// TwinCAT 3 PLC project XY_Motion_Control
// ProgramVersion: 3.1.4024.0
// libraries:
//   Tc2_Math, * (Beckhoff Automation GmbH)
//   Tc2_MC2, * (Beckhoff Automation GmbH)
//   Tc2_Standard, * (Beckhoff Automation GmbH)
//   Tc2_System, * (Beckhoff Automation GmbH)
//   Tc3_Module, * (Beckhoff Automation GmbH)
// project tree:
//   DUTs/ E_AutoSeqState.TcDUT, ST_MotionStep.TcDUT
//   / GlobalTextList.TcGTLO, PlcTask.TcTTO, Visualization Manager.TcVMO (not stored)
//   GVLs/ GVL_Motion.TcGVL
//   POUs/ AutoSequence.TcPOU, FB_XYZ_Movement.TcPOU, MAIN.TcPOU
//   VISUs/ Visualization.TcVIS
// real-time tasks:
//   TASK PlcTask: cycle T#10ms, priority 20, ADS port 350
// motion (NC):
//   TASK NC-Task 1 SAF: cycle T#2ms, priority 4, ADS port 501
//   TASK NC-Task 1 SVB: cycle T#10ms, priority 8, ADS port 511
//   AXIS Axis 1 (X) (id 1) // This is the X axis
//     Velo: RefSearch=3, SlowManual=5, FastManual=50
//     OtherSettings: AllowMotionCmdToSlave=true
//     encoder EncType=19
//       EncPara: ScaleFactorNumerator=3.8147e-05, MaxCount=#xffffffff
//         SoftEndMinControl: Enable=true, Range=-0.1
//         SoftEndMaxControl: Enable=true, Range=9.9
//         Inc: RefSoftSyncMask=#xffffffff
//     drive DrvType=16
//       DrvPara: MaxCount=#xffffffff, DriveControlDWord=#x00020100
//         Analog: TorqueSetpointScale=10, ScaleFactorActTorque=0.1
//         TimeComp: TaskDelayCycles=1
//     controller CtrType=1
//       CtrPara: PriorControlFactor=1
//         Observer: BandWidth=20
//   AXIS Axis 2 (Y) (id 2) // This is the Y axis
//     Velo: RefSearch=3, SlowManual=10, FastManual=50
//     OtherSettings: AllowMotionCmdToSlave=true
//     encoder EncType=19
//       EncPara: MaxCount=#xffffffff
//         SoftEndMinControl: Enable=true, Range=-34
//         SoftEndMaxControl: Enable=true
//         Inc: RefSoftSyncMask=#xffffffff
//     drive DrvType=16
//       DrvPara: MaxCount=#xffffffff, DriveControlDWord=#x00020100
//         Analog: TorqueSetpointScale=10, ScaleFactorActTorque=0.1
//         TimeComp: TaskDelayCycles=1
//     controller CtrType=1
//       CtrPara: PriorControlFactor=1
//         Observer: BandWidth=20
// I/O:
//   DEVICE Device 1 (Profinet Device CCAT (RT)) (disabled), AmsNetId 5.55.247.106.2.1
//   DEVICE Device 2 (EtherCAT), AmsNetId 5.55.247.106.3.1
//     Term 1 (EK1200) [EK1200-5000 EtherCAT Power supply (2A E-Bus)]
//       Term 2 (EL1008) [EL1008 8Ch. Dig. Input 24V, 3ms]
//       Term 3 (EL2008) [EL2008 8Ch. Dig. Output 24V, 0.5A]
//       Term 4 (EL9011) [EL9011 End Terminal]
//   DEVICE Device 5 (EtherCAT), AmsNetId 5.55.247.106.6.1
//     Drive 5 (R88D-KN01H-ECT) [R88D-KN01H-ECT G5 Series ServoDrive/Motor]
//     Drive 6 (R88D-KN01H-ECT) [R88D-KN01H-ECT G5 Series ServoDrive/Motor]
//   DEVICE Device 3 (NOV-DP-RAM)
// variable links:
//   NC-Task 1 SAF/Axes/Axis 1 (X) <-> Device 5 (EtherCAT)/Drive 5 (R88D-KN01H-ECT)
//     Drive/Inputs/In/nDataIn1 <-> 258th transmit PDO Mapping/Following error actual value
//     Drive/Inputs/In/nDataIn3[0] <-> 258th transmit PDO Mapping/Torque actual value
//     Drive/Inputs/In/nDcOutputTime <-> InfoData/DcOutputShift
//     Drive/Inputs/In/nState1 <-> 258th transmit PDO Mapping/Statusword
//     Drive/Inputs/In/nState2 <-> 258th transmit PDO Mapping/Statusword @bit 8
//     Drive/Inputs/In/nState4 @bit 1 <-> WcState/InputToggle
//     Drive/Inputs/In/nState4 <-> WcState/WcState
//     Drive/Outputs/Out/nCtrl1 <-> 258th receive PDO Mapping/Controlword
//     Drive/Outputs/Out/nCtrl2 <-> 258th receive PDO Mapping/Controlword @bit 8
//     Drive/Outputs/Out/nDataOut1 <-> 258th receive PDO Mapping/Target position
//     Enc/Inputs/In/nDataIn1 <-> 258th transmit PDO Mapping/Position actual value
//     Enc/Inputs/In/nDataIn3 <-> 258th transmit PDO Mapping/Touch probe pos1 pos value
//     Enc/Inputs/In/nDataIn5 <-> 258th transmit PDO Mapping/Touch probe pos2 pos value
//     Enc/Inputs/In/nDcInputTime <-> InfoData/DcInputShift
//     Enc/Inputs/In/nState4 @bit 1 <-> WcState/InputToggle
//     Enc/Inputs/In/nState4 <-> WcState/WcState
//     Enc/Inputs/In/nState5 <-> 258th transmit PDO Mapping/Touch probe status
//     Enc/Inputs/In/nState6 <-> 258th transmit PDO Mapping/Touch probe status @bit 8
//     Enc/Outputs/Out/nCtrl5 <-> 258th receive PDO Mapping/Touch probe function
//     Enc/Outputs/Out/nCtrl6 <-> 258th receive PDO Mapping/Touch probe function @bit 8
//   NC-Task 1 SAF/Axes/Axis 2 (Y) <-> Device 5 (EtherCAT)/Drive 6 (R88D-KN01H-ECT)
//     Drive/Inputs/In/nDataIn1 <-> 258th transmit PDO Mapping/Following error actual value
//     Drive/Inputs/In/nDataIn3[0] <-> 258th transmit PDO Mapping/Torque actual value
//     Drive/Inputs/In/nDcOutputTime <-> InfoData/DcOutputShift
//     Drive/Inputs/In/nState1 <-> 258th transmit PDO Mapping/Statusword
//     Drive/Inputs/In/nState2 <-> 258th transmit PDO Mapping/Statusword @bit 8
//     Drive/Inputs/In/nState4 @bit 1 <-> WcState/InputToggle
//     Drive/Inputs/In/nState4 <-> WcState/WcState
//     Drive/Outputs/Out/nCtrl1 <-> 258th receive PDO Mapping/Controlword
//     Drive/Outputs/Out/nCtrl2 <-> 258th receive PDO Mapping/Controlword @bit 8
//     Drive/Outputs/Out/nDataOut1 <-> 258th receive PDO Mapping/Target position
//     Enc/Inputs/In/nDataIn1 <-> 258th transmit PDO Mapping/Position actual value
//     Enc/Inputs/In/nDataIn3 <-> 258th transmit PDO Mapping/Touch probe pos1 pos value
//     Enc/Inputs/In/nDataIn5 <-> 258th transmit PDO Mapping/Touch probe pos2 pos value
//     Enc/Inputs/In/nDcInputTime <-> InfoData/DcInputShift
//     Enc/Inputs/In/nState4 @bit 1 <-> WcState/InputToggle
//     Enc/Inputs/In/nState4 <-> WcState/WcState
//     Enc/Inputs/In/nState5 <-> 258th transmit PDO Mapping/Touch probe status
//     Enc/Inputs/In/nState6 <-> 258th transmit PDO Mapping/Touch probe status @bit 8
//     Enc/Outputs/Out/nCtrl5 <-> 258th receive PDO Mapping/Touch probe function
//     Enc/Outputs/Out/nCtrl6 <-> 258th receive PDO Mapping/Touch probe function @bit 8
//   XY_Motion_Control/Motion_Control <-> Device 2 (EtherCAT)/Term 1 (EK1200)/Term 2 (EL1008)
//     PlcTask Inputs/GVL_Motion.bSensor_X <-> Channel 1/Input
//     PlcTask Inputs/GVL_Motion.bSensor_Y <-> Channel 3/Input
//   XY_Motion_Control/Motion_Control <-> Device 2 (EtherCAT)/Term 1 (EK1200)/Term 3 (EL2008)
//     PlcTask Outputs/GVL_Motion.bZlifter <-> Channel 2/Output
//   XY_Motion_Control/Motion_Control <-> NC-Task 1 SAF/Axes/Axis 1 (X)
//     PlcTask Inputs/GVL_Motion.Axis1.NcToPlc <-> Outputs/ToPlc
//     PlcTask Outputs/GVL_Motion.Axis1.PlcToNc <-> Inputs/FromPlc
//   XY_Motion_Control/Motion_Control <-> NC-Task 1 SAF/Axes/Axis 2 (Y)
//     PlcTask Inputs/GVL_Motion.Axis2.NcToPlc <-> Outputs/ToPlc
//     PlcTask Outputs/GVL_Motion.Axis2.PlcToNc <-> Inputs/FromPlc

CONFIGURATION XY_Motion_Control
    RESOURCE PLC ON TwinCAT3
        TASK PlcTask(INTERVAL := T#10ms, PRIORITY := 20);
        PROGRAM MAIN WITH PlcTask : MAIN;
    END_RESOURCE
END_CONFIGURATION

// ---- DUTs/E_AutoSeqState.TcDUT
{attribute 'qualified_only'}
{attribute 'strict'}
// Moves for the auto sequence
// Auto sekvenssin liikkeet
TYPE E_AutoSeqState :
(
	INIT,
    MOVE_X_SAFE_HOME,
	WAIT_X_SAFE_HOME,

    SET_Z_POSITION,
    WAIT_Z_DELAY,

    DECIDE_MOVE_ORDER,
	MOVE_Y,
    WAIT_Y,

    MOVE_X,
    WAIT_X,

    NEXT_STEP,

    PREPARE_RETURN_HOME,
    RETURN_HOME

);
END_TYPE

// ---- DUTs/ST_MotionStep.TcDUT
TYPE ST_MotionStep :
STRUCT
	fTargetX		: LREAL; // Target position of X axis - AXIS1, X axis kohde asento
	fTargetY		: LREAL; // Target position of Y axis - AXIS2, Y axis kohde asento
	nZaction		: INT; 	 // 1 = Lift, 2 = Lower, 0 = Do nothing, nostimen asennot
END_STRUCT
END_TYPE

// ---- GVLs/GVL_Motion.TcGVL
{attribute 'qualified_only'}
{attribute 'qualified_only'}
VAR_GLOBAL
	// Author RL
	// Hardware axis references
	// Axis viittaukset
	Axis1               : AXIS_REF;	// X
	Axis2               : AXIS_REF;	// Y
	
	// Core system control
	bEnableAll          : BOOL := TRUE;		// Enables the servo drives, aktivoi servot
	bResetAll           : BOOL := FALSE;	// Resets possible servo errors, resetoi servo viat
	bManualModeActive   : BOOL := FALSE; 	// Enables manual driving, aktivoi manualiajon
	
	// Homing inputs and status check after homing
	// Kotiutus inputit ja tarkistus kotiutuksen jälkeen
	bSensor_X           AT %I* : BOOL; 
	bSensor_Y           AT %I* : BOOL;
	bStartHoming        : BOOL := FALSE; 
	bXHomed             : BOOL := FALSE; 
	bYHomed             : BOOL := FALSE; 

	// Live axis position
	// Live axis asennot
	fCurrentX           : LREAL := 0.0;
	fCurrentY           : LREAL := 0.0;

	// "Z Axis" not really but kinda acts as a Z axis, this is a pneumatic lifter that is sitting on the Y axis
	// "Z Axis" Paineilma nostin Y akselin päällä
	bZlifter            AT %Q* : BOOL;      // FALSE = Raised, TRUE = Lowered)
	bZlifterManual		: BOOL;
	
	// Controls for manual driving, "Jogging"
	// Manuaaliajon kontrollit
	bJogForwardX        : BOOL := FALSE;    
	bJogForwardY        : BOOL := FALSE;    
	bJogBackwardsX      : BOOL := FALSE;    
	bJogBackwardsY      : BOOL := FALSE;
	fVelocityX          : LREAL := 5.0;
	fVelocityY          : LREAL := 10.0;
	
	// These calculate if moving is allowed, based on current position
	// Liikkumisen luvat, nykyisen sijainnin mukaan
	bX_Allow_Positive   : BOOL := FALSE;
	bX_Allow_Negative   : BOOL := FALSE;
	bY_Allow_Positive   : BOOL := FALSE;
	bY_Allow_Negative   : BOOL := FALSE;
	
	// States
	// Z nostimen tilat
	Z_IDLE          : INT := 0;
	Z_UP            : INT := 1;
	Z_DOWN          : INT := 2;
	
	iAutoState          : INT := 0; 
	bStartAutoseq     	: BOOL := FALSE;
	bAutoseqDone     	: BOOL := FALSE;
	bSequenceRunning	: BOOL;
	bRetrievalMode    	: BOOL := FALSE;  // FALSE = Put away pallets, TRUE = Take away pallets / Autosekvenssin Z lifter käänteiset tilat
	
	bExecuteMoveX    : BOOL;
    bExecuteMoveY    : BOOL;
    fTargetX         : LREAL;
    fTargetY         : LREAL;

	
	iStepPointer        : INT := 1;
	eSubPhase           : E_AutoSeqState := E_AutoSeqState.INIT;
	iTotalSteps         : INT := 9;
	
	// Go to config if u change these settings
	// This array system holds inside coordinates for the automatic sequence driving
	// Actions of the pneumatic lift are reversed when bRetrievalMode = TRUE
	// Automaattisen sekvenssin koordinaatit
	// Lifterin aktionit päinvaistaiset kun bRetrievalMode = TRUE
	astPath : ARRAY[1..9] OF ST_MotionStep := [
		// "Shelf 1" cycle
		
		(fTargetX := 2.8000, fTargetY := -0.6247,  nZAction := 1), // 2. Moce Y to shelf 1 height
		(fTargetX := 9.3720, fTargetY := -0.6247,  nZAction := 2), // 3. Drive in and lower forks
		(fTargetX := 2.8000, fTargetY := -0.6247,  nZAction := 1), // 4. Retreat to safe line and raise forks
		
		// "Shelf 2" cycle
		(fTargetX := 2.8000, fTargetY := -9.5381,	nZAction := 0), // 5. Drop Y to shelf 2 height
		(fTargetX := 9.3720, fTargetY := -9.5381,	nZAction := 2), // 6. Drive in and lower forks
		(fTargetX := 2.8000, fTargetY := -9.5381,	nZAction := 1), // 7. Retreat to safe line and raise forks
		
		// "Shelf 3" cycle
		(fTargetX := 2.8000, fTargetY := -18.7514,	nZAction := 0), // 8. Drop Y to shelf 3 height
		(fTargetX := 9.3720, fTargetY := -18.7514,	nZAction := 2), // 9. Drive in and lower forks
		(fTargetX := 0.0,	 fTargetY := -18.7514,	nZAction := 1)	// 10. Drive X out to 0 keep Y still
		
		
		// The auto sequence automatically handles moving X and Y back to 0.0 after this step	
	];
	
END_VAR

// ---- POUs/MAIN.TcPOU
// Author RL
PROGRAM MAIN
VAR
	XYZ	: FB_XYZ_Movement;
END_VAR

// Execute the entire system
AutoSequence();

XYZ(Axis1 := GVL_Motion.Axis1, Axis2 := GVL_Motion.Axis2);

END_PROGRAM

// ---- POUs/FB_XYZ_Movement.TcPOU
FUNCTION_BLOCK FB_XYZ_Movement
VAR_IN_OUT
    // Axis references
    Axis1                : AXIS_REF; // X
    Axis2                : AXIS_REF; // Y
END_VAR
VAR
    // Hardware Power and Reset Blocks
    fbPower1             : MC_Power;
    fbPower2             : MC_Power;
	
    fbReset1             : MC_Reset;
    fbReset2             : MC_Reset;
    
    // Core Motion Instances
    fbAutoMoveX          : MC_MoveAbsolute;
    fbAutoMoveY          : MC_MoveAbsolute;
	
    fbDriveToSensorX     : MC_MoveVelocity;
    fbDriveToSensorY     : MC_MoveVelocity;
	
    fbStopX              : MC_Stop;
    fbStopY              : MC_Stop;
	
    fbLockZeroX          : MC_SetPosition;
    fbLockZeroY          : MC_SetPosition;
	
    fbJogX               : MC_Jog;
    fbJogY               : MC_Jog;
	
	//Safety position reference
	fActPosX				 : LREAL;
	fActPosY				 : LREAL;
END_VAR

// Safety first, position reference form axis
// Paikan haku
fActPosX	:= Axis1.NcToPlc.ActPos;
fActPosY	:= Axis2.NcToPlc.ActPos;
THIS^.M_UpdateSafety();

// Axis Power, directional enables based on position
// Axis teho, luvat liike suunnille sijainnin perusteella
// X Axis 1
fbPower1(
    Axis            := Axis1, 
    Enable          := GVL_Motion.bEnableAll, 
    Enable_Positive := GVL_Motion.bEnableAll AND GVL_Motion.bX_Allow_Positive, 
    Enable_Negative := GVL_Motion.bEnableAll AND GVL_Motion.bX_Allow_Negative
);
// Y Axis 2
fbPower2(
    Axis            := Axis2, 
    Enable          := GVL_Motion.bEnableAll, 
    Enable_Positive := GVL_Motion.bEnableAll AND GVL_Motion.bY_Allow_Positive, 
    Enable_Negative := GVL_Motion.bEnableAll AND GVL_Motion.bY_Allow_Negative
);

// NC Kernel Error Resets
// Axis error resetit
fbReset1(
	Axis := Axis1,
	Execute := GVL_Motion.bResetAll);
	
fbReset2(
	Axis := Axis2,
	Execute := GVL_Motion.bResetAll);

IF GVL_Motion.bResetAll THEN
    GVL_Motion.bResetAll := FALSE;
END_IF

// Automated sequence, axis ref and enables, edit velocity if needed
// Automaattisen sekvenssin, axis viittaus ja luvat, tästä voi muutta automaattisen sekvenssin nopeutta halutessa
// Jos nopeutta on liikaa servo menee error tilaan (Set point karkaa liian kauas)
fbAutoMoveX(
    Axis     := Axis1, 
    Execute  := GVL_Motion.bExecuteMoveX AND NOT GVL_Motion.bManualModeActive, 
    Position := GVL_Motion.fTargetX, 
    Velocity := 10.0
);

fbAutoMoveY(
    Axis     := Axis2, 
    Execute  := GVL_Motion.bExecuteMoveY AND NOT GVL_Motion.bManualModeActive, 
    Position := GVL_Motion.fTargetY, 
    Velocity := 20.0
);


// Manual control, axis ref and enables
// Manuaali ajon axis viittaus, luvat
fbJogX(
    Axis         := Axis1,
    JogForward   := GVL_Motion.bJogForwardX AND GVL_Motion.bX_Allow_Positive AND GVL_Motion.bManualModeActive AND NOT GVL_Motion.bStartAutoseq,
    JogBackwards := GVL_Motion.bJogBackwardsX AND GVL_Motion.bX_Allow_Negative AND GVL_Motion.bManualModeActive AND NOT GVL_Motion.bStartAutoseq,
    Mode         := MC_JOGMODE_CONTINOUS,
    Velocity     := GVL_Motion.fVelocityX
);

fbJogY(
    Axis         := Axis2,
    JogForward   := GVL_Motion.bJogForwardY AND GVL_Motion.bY_Allow_Positive AND GVL_Motion.bManualModeActive AND NOT GVL_Motion.bStartAutoseq,
    JogBackwards := GVL_Motion.bJogBackwardsY AND GVL_Motion.bY_Allow_Negative AND GVL_Motion.bManualModeActive AND NOT GVL_Motion.bStartAutoseq,
    Mode         := MC_JOGMODE_CONTINOUS,
    Velocity     := GVL_Motion.fVelocityY
);

// Safety reset to turn off manual jogging if switched away from manual mode
// Manualiset liike komennot lakkaa, jos vaihdetaan kesken kaiken pois manuaali tilasta
IF NOT GVL_Motion.bManualModeActive THEN
    fbJogX(
		Axis := Axis1,
		JogForward := FALSE,
		JogBackwards := FALSE);
		
    fbJogY(
		Axis := Axis2,
		JogForward := FALSE,
		JogBackwards := FALSE);
END_IF

// Homing
// Kotiutus
fbDriveToSensorX(
	Axis := Axis1,
	Execute := GVL_Motion.bStartHoming,
	Velocity := 5.0,
	Direction := MC_Negative_Direction);
	
fbStopX(
	Axis := Axis1,
	Execute := GVL_Motion.bStartHoming AND GVL_Motion.bSensor_X);
	
fbLockZeroX(
	Axis := Axis1,
	Execute := GVL_Motion.bStartHoming AND fbStopX.Done,
	Position := 0.0);

fbDriveToSensorY(
	Axis := Axis2,
	Execute := GVL_Motion.bStartHoming,
	Velocity := 17.0,
	Direction := MC_Positive_Direction);
	
fbStopY(
	Axis := Axis2,
	Execute := GVL_Motion.bStartHoming AND GVL_Motion.bSensor_Y);
	
fbLockZeroY(
	Axis := Axis2,
	Execute := GVL_Motion.bStartHoming AND fbStopY.Done,
	Position := 0.0);

// Homing indication
// Kotiutuksen indikointi
IF fbLockZeroX.Done THEN 
    GVL_Motion.bXHomed := TRUE;
END_IF

IF fbLockZeroY.Done THEN
    GVL_Motion.bYHomed := TRUE;
END_IF

// Reset Homing when done
// Resetoidaan kotiutus kun se on valmis
IF GVL_Motion.bXHomed AND GVL_Motion.bYHomed THEN
    GVL_Motion.bStartHoming := FALSE;
END_IF

// Reset homing executions, so that homing can be done again if needed
// Resetoidaan kotiutus, jos tarvitaan uudestaan kotiuttaa
IF NOT GVL_Motion.bStartHoming THEN
    fbDriveToSensorX(
		Axis := Axis1,
		Execute := FALSE);
		
    fbStopX(
		Axis := Axis1,
		Execute := FALSE);
		
    fbLockZeroX(
		Axis := Axis1,
		Execute := FALSE);
    
    fbDriveToSensorY(
		Axis := Axis2,
		Execute := FALSE);
    
	fbStopY(
		Axis := Axis2, 
		Execute := FALSE);
    
	fbLockZeroY(
		Axis := Axis2,
		Execute := FALSE);
END_IF

// Author RL
METHOD PRIVATE M_UpdateSafety
VAR_INPUT
END_VAR
//Author RL
// System position
// Systeemin sijainti
GVL_Motion.fCurrentX := fActPosX;
GVL_Motion.fCurrentY := fActPosY;

IF GVL_Motion.bSequenceRunning THEN
    GVL_Motion.bManualModeActive := FALSE;
END_IF

IF GVL_Motion.bStartHoming THEN
    // During homing all movement is allowed
	// Kotiutuksen aikana kaikki liikesuunnan sallittu
    GVL_Motion.bX_Allow_Negative := TRUE; 
    GVL_Motion.bX_Allow_Positive := TRUE;
    GVL_Motion.bY_Allow_Negative := TRUE; 
    GVL_Motion.bY_Allow_Positive := TRUE;
END_IF
	
IF GVL_Motion.bManualModeActive THEN
	// Different safety limits for manual driving, this is to prevent hitting the shelves with forks in manual mode.
	// These are editable from here, but not recommended to ensure safe operation
	// Manuaaliajolla eri turvarajat, voi muutta, mutta ei suositeltu
	GVL_Motion.bX_Allow_Negative := (GVL_Motion.fCurrentX > -0.1);
    GVL_Motion.bX_Allow_Positive := (GVL_Motion.fCurrentX < 5.820);	// Note X is allowed to travell less in manual to protect possible forks/ Z lifter
                                       
    GVL_Motion.bY_Allow_Negative := (GVL_Motion.fCurrentY > -34.0);
   	GVL_Motion.bY_Allow_Positive := (GVL_Motion.fCurrentY < 0.0);
	
	GVL_Motion.bZlifter := GVL_Motion.bZlifterManual;	// Manual control for Z lifter, manuaaliset kontrollit Z lifterille
END_IF

IF GVL_Motion.bSequenceRunning THEN
	// Safety limits for automatic sequence
	// These same values are also in the AXIS settings under parameter - limit switches
	// These values are safe operation boundaries so that we dont crash the lifter/forks in to the shelves
	// If you wish to edit these, go under Axis -> Parameters -> Limit switches
	// Auto sekvenssin turvarajat, nämä on myös asetettu suoraan molempiin Axiksiin niiden asetuksista
    GVL_Motion.bX_Allow_Negative := (GVL_Motion.fCurrentX > -0.1);
    GVL_Motion.bX_Allow_Positive := (GVL_Motion.fCurrentX < 9.9);
                                        
    GVL_Motion.bY_Allow_Negative := (GVL_Motion.fCurrentY > -34.0);
    GVL_Motion.bY_Allow_Positive := (GVL_Motion.fCurrentY < 0.0);
END_IF
END_METHOD

END_FUNCTION_BLOCK

// ---- POUs/AutoSequence.TcPOU
// Author RL
PROGRAM AutoSequence
VAR
    bSequenceResetPulse : BOOL;
    tPneumaticDelay     : TON;
    bOldZlifter         : BOOL;
	bSequenceRunning	: BOOL;
END_VAR

// Author RL
IF GVL_Motion.bStartAutoseq AND GVL_Motion.bXHomed AND GVL_Motion.bYHomed AND NOT GVL_Motion.bSequenceRunning THEN
    GVL_Motion.bStartAutoseq    := FALSE; // Switches HMI button to FALSE, Laittaa HMI nappulan FALSE
    GVL_Motion.bSequenceRunning := TRUE;  // True while sequence running, TRUE kun sekvenssi käynnissä
    GVL_Motion.bAutoseqDone     := FALSE; // FALSE while sequence active, FALSE kun sekvenssi käynnissä
	
	GVL_Motion.iStepPointer     := 1;     
    GVL_Motion.bExecuteMoveX    := FALSE; // Wipes old move triggers, pyyhkii vanhat executet
    GVL_Motion.bExecuteMoveY    := FALSE; // Wipes old move triggers, pyyhkii vanhat executet
	
    GVL_Motion.eSubPhase		:= E_AutoSeqState.INIT;
	
END_IF

// Auto Sequence / Automaattinen sekvenssi
IF GVL_Motion.bSequenceRunning THEN
    bSequenceResetPulse := FALSE;

    // Check if there are still valid steps left to run in path array
    // Tarkastetaan onko vielä askelia jäljellä
    IF GVL_Motion.iStepPointer <= GVL_Motion.iTotalSteps THEN
    
         CASE GVL_Motion.eSubPhase OF
			// Init
             E_AutoSeqState.INIT:
			 
                tPneumaticDelay(IN := FALSE);
				GVL_Motion.bExecuteMoveX := FALSE;
                GVL_Motion.bExecuteMoveY := FALSE;

             GVL_Motion.eSubPhase := E_AutoSeqState.MOVE_X_SAFE_HOME;
	
		// Pull X to home if not at home before changing Y position, this is to avoid possible collision
        // Vedetään X kotiin ennen Y:tä, näin vältetään mahdolliset törmäykset
        E_AutoSeqState.MOVE_X_SAFE_HOME:
	
			GVL_Motion.fTargetX := 0.0;
			GVL_motion.bExecuteMoveX := TRUE;
			
			GVL_Motion.eSubPhase := E_AutoSeqState.WAIT_X_SAFE_HOME;
        
		// Wait for X to move home before starting the sequence if X is not at home
		// Odotetaan että X liikkuu kotiin ennen aloitusta
		E_AutoSeqState.WAIT_X_SAFE_HOME:
		
			GVL_Motion.bExecuteMoveX := FALSE;
			
			IF ABS(GVL_Motion.fCurrentX) <= 0.05 AND NOT MAIN.XYZ.fbAutoMoveX.Busy THEN
				GVL_Motion.eSubPhase := E_AutoSeqState.SET_Z_POSITION;
			END_IF
		// Evaluate if the Z lifter needs to actuate for the current step
        // Arvioidaan tarvitaanko Z lifterin asentoa vaihtaa
        E_AutoSeqState.SET_Z_POSITION:
			
			bOldZlifter := GVL_Motion.bZlifter;
			
			// Different modes lifting and lowering
			// Eri modet nosto ja lasku
            IF NOT GVL_Motion.bRetrievalMode THEN
				IF GVL_Motion.astPath[GVL_Motion.iStepPointer].nZAction = GVL_Motion.Z_UP THEN
					GVL_Motion.bZlifter := FALSE; 
                ELSIF GVL_Motion.astPath[GVL_Motion.iStepPointer].nZAction = GVL_Motion.Z_DOWN THEN
                    GVL_Motion.bZlifter := TRUE; 
                END_IF
                ELSE
                    IF GVL_Motion.astPath[GVL_Motion.iStepPointer].nZAction = GVL_Motion.Z_UP THEN
                        GVL_Motion.bZlifter := TRUE; 
                    ELSIF GVL_Motion.astPath[GVL_Motion.iStepPointer].nZAction = GVL_Motion.Z_DOWN THEN
                        GVL_Motion.bZlifter := FALSE; 
                    END_IF
            END_IF
                
            IF GVL_Motion.bZlifter = bOldZlifter THEN
                    GVL_Motion.eSubPhase := E_AutoSeqState.DECIDE_MOVE_ORDER; 
                ELSE
                    GVL_Motion.eSubPhase := E_AutoSeqState.WAIT_Z_DELAY; 
            END_IF
            
			// 1 sec delay after Z moves to avoid unwanted disasters
            // 1 sekuntin viive, jotta Z liikkeet ei tapahdu samanaikaisesti Y/X liikkeiten kanssa 
            E_AutoSeqState.WAIT_Z_DELAY:
			
                tPneumaticDelay(IN := TRUE, PT := T#1000MS);
				
                IF tPneumaticDelay.Q THEN 
                    tPneumaticDelay(IN := FALSE); 
                    GVL_Motion.eSubPhase := E_AutoSeqState.DECIDE_MOVE_ORDER; 
                END_IF
				
            // Decide which moves to make next
            // Tulevien liikkeiten valinta
			E_AutoSeqState.DECIDE_MOVE_ORDER:
			
				GVL_Motion.bExecuteMoveX	:= FALSE;
				GVL_Motion.bExecuteMoveY	:= FALSE;
				
                IF GVL_Motion.astPath[GVL_Motion.iStepPointer].fTargetX = 0.0 THEN
					
                    IF ABS(GVL_Motion.fCurrentX - GVL_Motion.astPath[GVL_Motion.iStepPointer].fTargetX) > 0.05 THEN
                        GVL_Motion.fTargetX := GVL_Motion.astPath[GVL_Motion.iStepPointer].fTargetX; 
                        GVL_Motion.fTargetY := GVL_Motion.fCurrentY; 
                        GVL_Motion.bExecuteMoveX := TRUE;
						GVL_Motion.eSubPhase := E_AutoSeqState.WAIT_X;
					ELSE
						GVL_Motion.eSubPhase := E_AutoSeqState.MOVE_Y;
					END_IF
                        
                    ELSE
						IF ABS(GVL_Motion.fCurrentY - GVL_motion.astPath[GVL_Motion.iStepPointer].fTargetY) > 0.05 THEN
							GVL_motion.eSubPhase := E_AutoSeqState.MOVE_Y;
						ELSE
							GVL_Motion.eSubPhase := E_AutoSeqState.MOVE_X;
						END_IF
				END_IF
				
			// Set targets and move Y
			// Asetetaan kohde ja liikutetaan Y	
			E_AutoSeqState.MOVE_Y:
				
				GVL_Motion.fTargetX := GVL_Motion.fCurrentX; 
                GVL_Motion.fTargetY := GVL_Motion.astPath[GVL_Motion.iStepPointer].fTargetY;
                GVL_Motion.bExecuteMoveX := FALSE; 
                GVL_Motion.bExecuteMoveY := TRUE;
						
			GVL_Motion.eSubPhase := E_AutoSeqState.WAIT_Y;
			
			// Wait for Y to be done with moving before moving X
			// Odotetaan kunnes Y on valmis ennen kuin liikutetaan X
			E_AutoSeqState.WAIT_Y:
				
				IF ABS(GVL_Motion.fCurrentY - GVL_Motion.astPath[GVL_Motion.iStepPointer].fTargetY) <= 0.05 AND NOT MAIN.XYZ.fbAutoMoveY.Busy THEN
					GVL_Motion.bExecuteMoveY := FALSE;
							
					IF GVL_Motion.astPath[GVL_Motion.iStepPointer].fTargetX = 0.0 THEN
						GVL_Motion.eSubPhase := E_AutoSeqState.NEXT_STEP;
						ELSE
							GVL_Motion.eSubPhase := E_AutoSeqState.MOVE_X;
					END_IF
				END_IF
				
			// Set targets and move X
			// Asetetaan kohde ja liikutetaan X			
			E_AutoSeqState.MOVE_X :
				
                GVL_Motion.fTargetX := GVL_Motion.astPath[GVL_Motion.iStepPointer].fTargetX; 
                GVL_Motion.fTargetY := GVL_Motion.fCurrentY;
                GVL_Motion.bExecuteMoveX := TRUE; 
                GVL_Motion.bExecuteMoveY := FALSE;
						
			GVL_Motion.eSubPhase := E_AutoSeqState.WAIT_X;
			
			// Wait for X to be done with moving before moving Y
			// Odotetaan kunnes X on valmis ennen kuin liikutetaan Y		
			E_AutoSeqState.WAIT_X:
				
				IF ABS(GVL_Motion.fCurrentX - GVL_Motion.astPath[GVL_Motion.iStepPointer].fTargetX) <= 0.05 AND NOT MAIN.XYZ.fbAutoMoveX.Busy THEN
					GVL_Motion.bExecuteMoveX := FALSE;
							
					IF GVL_motion.astPath[GVL_Motion.iStepPointer].fTargetX = 0.0 THEN
						GVL_Motion.eSubPhase := E_AutoSeqState.MOVE_Y;
						ELSE
							GVL_Motion.eSubPhase := E_AutoSeqState.NEXT_STEP;
					END_IF
				END_IF
			
			//Both axes in position evaluate where to go next
			// Molemmat axes oikeissa paikoissa arvioi mihin mennään seuraavaksi			
			E_AutoSeqState.NEXT_STEP:
				
				IF GVL_Motion.iStepPointer = GVL_motion.iTotalSteps THEN
					GVL_Motion.eSubPhase := E_AutoSeqState.PREPARE_RETURN_HOME;
				ELSE
					GVL_Motion.iStepPointer := GVL_Motion.iStepPointer +1;
							
					IF  GVL_Motion.astPath[GVL_Motion.iStepPointer].nZaction = 0 THEN
						GVL_Motion.eSubPhase := E_AutoSeqState.DECIDE_MOVE_ORDER;
					ELSE
						GVL_Motion.eSubPhase := E_AutoSeqState.SET_Z_POSITION;
					END_IF
				END_IF
			
			// Prepare returning to home after finishing sequence
			// Valmistellaan kotiin paluu kun sekvenssi on valmis
			E_AutoSeqState.PREPARE_RETURN_HOME:
			
				GVL_Motion.bExecuteMoveX := FALSE;
				GVL_Motion.bExecuteMoveY := FALSE;
				
				GVL_Motion.fTargetX := 0.0;
                GVL_Motion.fTargetY := 0.0;

                GVL_Motion.bExecuteMoveY := TRUE;
				
			GVL_Motion.eSubPhase	 := E_AutoSeqState.RETURN_HOME;
			
			// Return home
			// Paluu kotiin 
            E_AutoSeqState.RETURN_HOME:
                       
             	IF MAIN.XYZ.fbAutoMoveY.Busy THEN
					GVL_Motion.bExecuteMoveY := FALSE;
                END_IF
				
   				IF ABS(GVL_Motion.fCurrentX) <= 0.05
                    AND ABS(GVL_Motion.fCurrentY) <= 0.05
                    AND NOT MAIN.XYZ.fbAutoMoveX.Busy
                    AND NOT MAIN.XYZ.fbAutoMoveY.Busy THEN

                    GVL_Motion.bExecuteMoveX := FALSE;
                    GVL_Motion.bExecuteMoveY := FALSE;

                    GVL_Motion.bZlifter := NOT GVL_Motion.bRetrievalMode;

                    GVL_Motion.bAutoseqDone     := TRUE;
                    GVL_Motion.bSequenceRunning := FALSE;
                    GVL_Motion.bStartAutoseq    := FALSE;

                    GVL_Motion.iStepPointer     := 1;
                    GVL_Motion.eSubPhase        := E_AutoSeqState.INIT;
                END_IF
				ELSE
    				GVL_Motion.eSubPhase := E_AutoSeqState.INIT;
          END_CASE
    END_IF
ELSE
    GVL_Motion.bExecuteMoveX := FALSE; 
    GVL_Motion.bExecuteMoveY := FALSE; 
    tPneumaticDelay(IN := FALSE);
    
    // Variable is ALWAYS forced to false when idle
    // Idlenä aina FALSE
    GVL_Motion.bStartAutoseq := FALSE; 
    
    IF NOT GVL_Motion.bAutoseqDone THEN
        bSequenceResetPulse := TRUE;
    ELSE
        bSequenceResetPulse := FALSE;
    END_IF
END_IF

END_PROGRAM

// ---- GlobalTextList.TcGTLO
TEXTLIST GlobalTextList
  401 = 'Allow X Negative'
  178 = 'Allow X Positive'
  504 = 'Allow Y Negative'
  962 = 'Allow Y Positive'
  920 = 'Auto Seq'
  348 = 'Axis 1 (X) Homed'
  783 = 'Axis 2 (Y) Homed'
  39 = 'Enable All'
  136 = 'Homing'
  613 = 'Jog X Backwards'
  374 = 'Jog X forward'
  551 = 'Jog Y Backwards'
  287 = 'Jog Y forward'
  427 = 'Lift pallet'
  362 = 'Lifter UP/DOWN'
  747 = 'Lower lifter'
  111 = 'Lower pallet'
  91 = 'Manual Mode'
  282 = 'Raise lifter'
  616 = 'Reset All'
  777 = 'X axis manual speed'
  364 = 'Y axis manual speed'
END_TEXTLIST

// ---- VISUs/Visualization.TcVIS
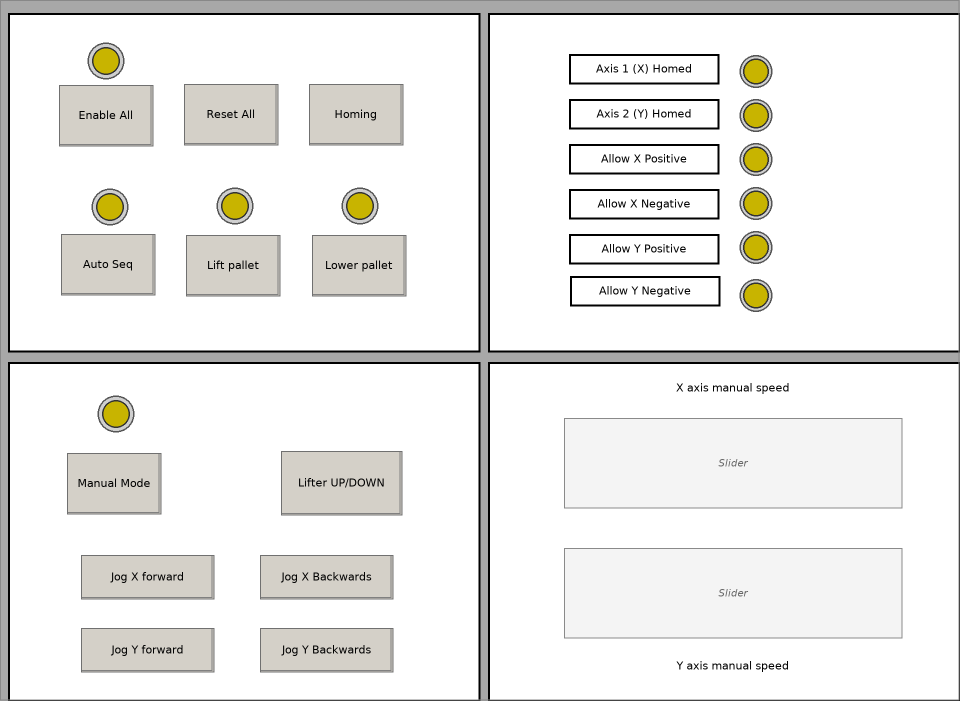
VISUALIZATION Visualization  // 960x701
    Rectangle (8,13 472x339)
    Rectangle (488,13 472x339)
    Rectangle (488,362 472x339)
    Rectangle (8,362 472x339)
    Button (59,85 94x61), "Enable All", colour toggle: GVL_Motion.bEnableAll, pressed state: GVL_Motion.bEnableAll
        OnMouseClick: toggle GVL_Motion.bEnableAll
    Button (184,84 94x61), "Reset All"
        tap GVL_Motion.bResetAll
        toggle GVL_Motion.bResetAll
    Button (67,453 94x61), "Manual Mode", pressed state: GVL_Motion.bManualModeActive
        OnMouseClick: toggle GVL_Motion.bManualModeActive
    Button (61,234 94x61), "Auto Seq", pressed state: GVL_Motion.bStartAutoseq
        OnMouseClick: toggle GVL_Motion.bStartAutoseq
    Button (309,84 94x61), "Homing", pressed state: GVL_Motion.bStartHoming
        toggle GVL_Motion.bStartHoming
    Lamp1 (85,40 42x42), variable: GVL_Motion.bEnableAll, style: Lamp-Lamp1-Yellow
    Lamp1 (95,393 42x42), variable: GVL_Motion.bManualModeActive, style: Lamp-Lamp1-Yellow
    Button (81,555 133x44), "Jog X forward", pressed state: GVL_Motion.bJogForwardX
        OnMouseDown: toggle GVL_Motion.bJogForwardX
        OnMouseUp: toggle GVL_Motion.bJogForwardX
    Button (260,555 133x44), "Jog X Backwards", pressed state: GVL_Motion.bJogBackwardsX
        OnMouseDown: toggle GVL_Motion.bJogBackwardsX
        OnMouseUp: toggle GVL_Motion.bJogBackwardsX
    Button (81,628 133x44), "Jog Y forward", pressed state: GVL_Motion.bJogForwardY
        OnMouseDown: toggle GVL_Motion.bJogForwardY
        OnMouseUp: toggle GVL_Motion.bJogForwardY
    Button (260,628 133x44), "Jog Y Backwards", pressed state: GVL_Motion.bJogBackwardsY
        OnMouseDown: toggle GVL_Motion.bJogBackwardsY
        OnMouseUp: toggle GVL_Motion.bJogBackwardsY
    Slider (564,418 338x90), variable: GVL_Motion.fVelocityX, scale 0..30
    Slider (564,548 338x90), variable: GVL_Motion.fVelocityY, scale 0..30
    Lamp1 (737,52 38x39), variable: GVL_Motion.bXHomed, style: Lamp-Lamp1-Yellow
    Lamp1 (737,96 38x39), variable: GVL_Motion.bYHomed, style: Lamp-Lamp1-Yellow
    Lamp1 (737,140 38x39), variable: GVL_Motion.bX_Allow_Positive, style: Lamp-Lamp1-Yellow
    Lamp1 (737,184 38x39), variable: GVL_Motion.bX_Allow_Negative, style: Lamp-Lamp1-Yellow
    Lamp1 (737,228 38x39), variable: GVL_Motion.bY_Allow_Positive, style: Lamp-Lamp1-Yellow
    Lamp1 (737,276 38x39), variable: GVL_Motion.bY_Allow_Negative, style: Lamp-Lamp1-Yellow
    Lamp1 (89,186 42x42), variable: GVL_Motion.bSequenceRunning, style: Lamp-Lamp1-Yellow
    Button (186,235 94x61), "Lift pallet", pressed state: GVL_Motion.bRetrievalMode
        OnMouseClick: execute { GVL_Motion.bRetrievalMode := TRUE; }
    Button (312,235 94x61), "Lower pallet", pressed state: NOT GVL_Motion.bRetrievalMode
        OnMouseClick: execute { GVL_Motion.bRetrievalMode := FALSE; }
    Lamp1 (214,185 42x42), variable: GVL_Motion.bRetrievalMode, style: Lamp-Lamp1-Yellow
    Lamp1 (339,185 42x42), variable: NOT GVL_Motion.bRetrievalMode, style: Lamp-Lamp1-Yellow
    Rectangle (570,276 150x30), "Allow Y Negative"
    Rectangle (569,234 150x30), "Allow Y Positive"
    Rectangle (569,189 150x30), "Allow X Negative"
    Rectangle (569,144 150x30), "Allow X Positive"
    Rectangle (569,99 150x30), "Axis 2 (Y) Homed"
    Rectangle (569,54 150x30), "Axis 1 (X) Homed"
    Button (281,451 121x64), "Lifter UP/DOWN", pressed state: GVL_Motion.bManualModeActive
        toggle GVL_Motion.bZlifterManual
    Label (658,373 150x30), "X axis manual speed"
    Label (658,651 150x30), "Y axis manual speed"
END_VISUALIZATION
